FUNCTION_BLOCK FB_EZylinder
VAR_INPUT
	bGate :BOOL;
	bError :BOOL;
END_VAR
VAR_OUTPUT
	bR1 :BOOL;
	bR2 :BOOL;
END_VAR
VAR
END_VAR

bR1 :=bGate;
bR2 := NOT bGate;

IF bError THEN
	bR1 := FALSE;
	bR2 := FALSE;
END_IF

END_FUNCTION_BLOCK

(* stored: Version 1.1.0.1, ProductVersion 3.1.4026.18
   POU FB_EZylinder: Id {5264cd30-3c9c-4c04-b81c-e07e59db338a}, SpecialFunc None *)
